// SIMATIC STEP 7 (V5.x) project tank-2pump-memory-exch
// CPU: CPU 312

SYMBOL_TABLE
"start"	I 0.0	BOOL
"stop"	I 0.1	BOOL
"empty sen"	I 0.2	BOOL
"full sen"	I 0.3	BOOL
"loop marker"	M 0.0	BOOL
"pump1 sit"	M 0.1	BOOL
"pump2 sit"	M 0.2	BOOL
"pump1"	Q 0.0	BOOL
"pump2"	Q 0.1	BOOL
END_SYMBOL_TABLE
